// TIA Portal V17 export
// export: Created 2025-06-25T13:13:25.5147908Z, ExportSetting WithDefaults, DisplayName Totally Integrated Automation Portal, DisplayVersion V17 Update 8, DisplayName TIA Portal Openness, DisplayVersion V17 Update 8, DisplayName TIA Portal Version Control Interface, DisplayVersion V17, DisplayName STEP 7 Professional, DisplayVersion V17 Update 8, DisplayName STEP 7 Safety, DisplayVersion V17 Update 6, DisplayName WinCC Advanced, DisplayVersion V17 Update 8
DATA_BLOCK "DB_Valves"   // DB46
{ S7_Optimized_Access := 'FALSE' }
AUTHOR : Heaten
VERSION : 0.1
// stored: AutoNumber false, DBAccessibleFromOPCUA true, DBAccessibleFromWebserver true, IsOnlyStoredInLoadMemory false, IsWriteProtectedInAS false
   VAR RETAIN
      HBL_HCV_576 : "stRegulatingValve";   // Expansion Valve A
      HBL_HCV_578 : "stRegulatingValve";   // Expansion Valve B
      HBL_HCV_577 { S7_SetPoint := 'True'} : "stRegulatingValve";   // Expansion Valve A2
      HBL_HCV_579 { S7_SetPoint := 'True'} : "stRegulatingValve";   // Expansion Valve B2
      HBL_HCV_515 { S7_SetPoint := 'True'} : "stRegulatingValve";   // Heat sink condensate blowdown flow control valve
      HBL_HCV_575 { S7_SetPoint := 'True'} : "stRegulatingValve";   // Recuperator oil drain valve
      HBL_HCV_616 { S7_SetPoint := 'True'} : "stRegulatingValve";   // Recuperator bypass valve
      HBL_HCV_700 { S7_SetPoint := 'True'} : "stRegulatingValve";   // Oil recovery refrigerant blowdown valve
      HBL_HCV_514 { S7_SetPoint := 'True'} : "stRegulatingValve";   // Heat sink discharge pressure control valve
      HBL_HCV_548 { S7_SetPoint := 'True'} : "stRegulatingValve";   // Heat source suction pressure control valve
      CPC_HCV_853 { S7_SetPoint := 'True'} : "stRegulatingValve";   // CPC cooler water control valve
      CPC_HCV_880 { S7_SetPoint := 'True'} : "stRegulatingValve";   // CPC subcooler water control valve
      HBL_HCV_900 { S7_SetPoint := 'True'} : "stRegulatingValve";   // Heat sink condensate feed valve
      HBL_HV_640 { S7_SetPoint := 'True'} : "stProcessValve2";   // Suction accumulator drain valve
      HBL_HV_670 { S7_SetPoint := 'True'} : "stProcessValve2";   // Discharge accumulator drain valve
      CPC_HV_852 { S7_SetPoint := 'True'} : "stProcessValve2";   // CPC cooler enable valve
      HBL_HV_861 { S7_SetPoint := 'True'} : "stProcessValve2";   // Compressor manifold drain valve
   END_VAR
BEGIN
   // HBL_HCV_576.Cmd.Position : Expansion Valve A
   HBL_HCV_576.Cmd.Position.Raw.iMax := 27648;
   HBL_HCV_576.Cmd.Position.Eng.fMin := 0.0;
   HBL_HCV_576.Cmd.Position.Eng.fMax := 100.0;
   // HBL_HCV_576.Stat.Position : Expansion Valve A
   HBL_HCV_576.Stat.Position.Raw.iMin := 0;
   HBL_HCV_576.Stat.Position.Raw.iMax := 27648;
   HBL_HCV_576.Stat.Position.Eng.fMin := 0.0;
   HBL_HCV_576.Stat.Position.Eng.fMax := 100.0;
   // HBL_HCV_578.Cmd.Position : Expansion Valve B
   HBL_HCV_578.Cmd.Position.Raw.iMin := 0;
   HBL_HCV_578.Cmd.Position.Raw.iMax := 27648;
   HBL_HCV_578.Cmd.Position.Eng.fMin := 0.0;
   HBL_HCV_578.Cmd.Position.Eng.fMax := 100.0;
   // HBL_HCV_578.Stat.Position : Expansion Valve B
   HBL_HCV_578.Stat.Position.Raw.iMin := 0;
   HBL_HCV_578.Stat.Position.Raw.iMax := 27648;
   HBL_HCV_578.Stat.Position.Eng.fMin := 0.0;
   HBL_HCV_578.Stat.Position.Eng.fMax := 100.0;
   HBL_HCV_577.Cmd.Position.Raw.iMin := 0;
   HBL_HCV_577.Cmd.Position.Raw.iMax := 27648;
   HBL_HCV_577.Cmd.Position.Eng.fMin := 0.0;
   HBL_HCV_577.Cmd.Position.Eng.fMax := 100.0;
   HBL_HCV_577.Stat.Position.Raw.iMin := 0;
   HBL_HCV_577.Stat.Position.Raw.iMax := 27648;
   HBL_HCV_577.Stat.Position.Eng.fMin := 0.0;
   HBL_HCV_577.Stat.Position.Eng.fMax := 100.0;
   HBL_HCV_579.Cmd.Position.Raw.iMin := 0;
   HBL_HCV_579.Cmd.Position.Raw.iMax := 27648;
   HBL_HCV_579.Cmd.Position.Eng.fMin := 0.0;
   HBL_HCV_579.Cmd.Position.Eng.fMax := 100.0;
   HBL_HCV_579.Stat.Position.Raw.iMin := 0;
   HBL_HCV_579.Stat.Position.Raw.iMax := 27648;
   HBL_HCV_579.Stat.Position.Eng.fMin := 0.0;
   HBL_HCV_579.Stat.Position.Eng.fMax := 100.0;
   HBL_HCV_515.Cmd.Position.Raw.iMin := 0;
   HBL_HCV_515.Cmd.Position.Raw.iMax := 27648;
   HBL_HCV_515.Cmd.Position.Eng.fMin := 0.0;
   HBL_HCV_515.Cmd.Position.Eng.fMax := 100.0;
   HBL_HCV_515.Stat.Position.Raw.iMin := 0;
   HBL_HCV_515.Stat.Position.Raw.iMax := 27648;
   HBL_HCV_515.Stat.Position.Eng.fMin := 0.0;
   HBL_HCV_515.Stat.Position.Eng.fMax := 100.0;
   HBL_HCV_575.Cmd.Position.Raw.iMin := 0;
   HBL_HCV_575.Cmd.Position.Raw.iMax := 27648;
   HBL_HCV_575.Cmd.Position.Eng.fMin := 0.0;
   HBL_HCV_575.Cmd.Position.Eng.fMax := 100.0;
   HBL_HCV_575.Stat.Position.Raw.iMin := 0;
   HBL_HCV_575.Stat.Position.Raw.iMax := 27648;
   HBL_HCV_575.Stat.Position.Eng.fMin := 0.0;
   HBL_HCV_575.Stat.Position.Eng.fMax := 100.0;
   HBL_HCV_616.Cmd.Position.Raw.iMin := 0;
   HBL_HCV_616.Cmd.Position.Raw.iMax := 27648;
   HBL_HCV_616.Cmd.Position.Eng.fMin := 0.0;
   HBL_HCV_616.Cmd.Position.Eng.fMax := 100.0;
   HBL_HCV_616.Stat.Position.Raw.iMin := 0;
   HBL_HCV_616.Stat.Position.Raw.iMax := 27648;
   HBL_HCV_616.Stat.Position.Eng.fMin := 0.0;
   HBL_HCV_616.Stat.Position.Eng.fMax := 0.0;
   HBL_HCV_700.Cmd.Position.Raw.iMin := 0;
   HBL_HCV_700.Cmd.Position.Raw.iMax := 27648;
   HBL_HCV_700.Cmd.Position.Eng.fMin := 0.0;
   HBL_HCV_700.Cmd.Position.Eng.fMax := 100.0;
   HBL_HCV_700.Stat.Position.Raw.iMin := 0;
   HBL_HCV_700.Stat.Position.Raw.iMax := 27648;
   HBL_HCV_700.Stat.Position.Eng.fMin := 0.0;
   HBL_HCV_700.Stat.Position.Eng.fMax := 100.0;
   HBL_HCV_548.Cmd.Position.Raw.iMin := 0;
   HBL_HCV_548.Cmd.Position.Raw.iMax := 27648;
   HBL_HCV_548.Cmd.Position.Eng.fMin := 0.0;
   HBL_HCV_548.Cmd.Position.Eng.fMax := 100.0;
   HBL_HCV_548.Stat.Position.Raw.iMin := 0;
   HBL_HCV_548.Stat.Position.Raw.iMax := 27648;
   HBL_HCV_548.Stat.Position.Eng.fMin := 0.0;
   HBL_HCV_548.Stat.Position.Eng.fMax := 100.0;
   CPC_HCV_853.Cmd.Position.Eng.fMax := 100.0;
   CPC_HCV_853.Stat.Position.Eng.fMax := 100.0;
   CPC_HCV_880.Cmd.Position.Eng.fMax := 100.0;
   CPC_HCV_880.Stat.Position.Eng.fMax := 100.0;
END_DATA_BLOCK
